// TIA Portal V16 export
// export: Created 2021-09-08T12:46:15.7751045Z, ExportSetting WithDefaults, DisplayName Totally Integrated Automation Portal, DisplayVersion V16 Update 3, DisplayName TIA Portal Version Control Interface, DisplayVersion V16 Update 2, DisplayName TIA Portal Openness, DisplayVersion V16 Update 3, DisplayName TIA Portal Teamcenter Gateway, DisplayVersion V16, DisplayName STEP 7 Professional, DisplayVersion V16 Update 3, DisplayName STEP 7 Safety, DisplayVersion V16, DisplayName WinCC Advanced, DisplayVersion V16 Update 3
TYPE "Av"
// stored: IsFailsafeCompliant false
   STRUCT
      mode : Bool;   // 0-ручной, 1-авто
      cmAuto { ExternalAccessible := 'False'; ExternalVisible := 'False'; ExternalWritable := 'False'} : Bool;   // авто команда
      cmHand : Bool;   // ручная команда
      block { ExternalAccessible := 'False'; ExternalVisible := 'False'; ExternalWritable := 'False'} : Bool;   // Внешняя блокировка
      error { ExternalAccessible := 'False'; ExternalVisible := 'False'; ExternalWritable := 'False'} : Bool;   // Общая ошибка
      checkOC { S7_SetPoint := 'True'} : Bool;   // Проверка концевиков
      outCmStart { ExternalAccessible := 'False'; ExternalVisible := 'False'; ExternalWritable := 'False'} : Bool;   // Программный выход
      st : Word;   // Состояние
      tOpen { S7_SetPoint := 'True'} : Int := 10;   // Время открытия, сек
      tClose { S7_SetPoint := 'True'} : Int := 10;   // Время закрытия, сек
      ack { ExternalAccessible := 'False'; ExternalVisible := 'False'; ExternalWritable := 'False'} : Word;
      spare_0 { ExternalAccessible := 'False'; ExternalVisible := 'False'; ExternalWritable := 'False'} : Word;
      spare_1 { ExternalAccessible := 'False'; ExternalVisible := 'False'; ExternalWritable := 'False'} : DInt;
   END_STRUCT;
END_TYPE
